Fanuc KAREL source: kb00150.KL

-- PROVISIONAL review KL for V1013-1; original PC SHA256 7e487c56d4365d8ae521bc3648a3ff10b0293b536462a349bf4bde1ced0e537b
-- Incomplete behavior may be omitted. Consult companion uncertainty JSON. Do not deploy.
PROGRAM KB00150
%NOLOCKGROUP
BEGIN
  -- UNRESOLVED_PC offsets 5-14; opcodes 3F,75
  -- UNRESOLVED_PC offsets 19-28; opcodes 3F,75
  -- UNRESOLVED_PC offsets 33-42; opcodes 3F,75
  -- UNRESOLVED_PC offsets 47-56; opcodes 3F,75
  -- UNRESOLVED_PC offsets 61-68; opcodes 9D,23
  -- UNRESOLVED_PC offsets 73-115; opcodes 27,22,2A,22,2A,22,2A,22,2A,22,31
  -- UNRESOLVED_PC offsets 120-124; opcodes 7F
END KB00150
